Fanuc KAREL source: Client.kl

PROGRAM TCP_Client

------------------------------------ TCP_Client Plug-In ------------------------------------
-- Author: Niccolo' Quadrani
-- Date: 9/05/2025
-- Version: 1.0.0
------------------------------------ TCP_Client Plug-In ------------------------------------


------------------------------------ Import ------------------------------------

%RWACCESS
%STACKSIZE = 4096
%NOLOCKGROUP
%NOBUSYLAMP
%NOPAUSE = ERROR + COMMAND + TPENABLE
%ENVIRONMENT uif
%ENVIRONMENT sysdef
%ENVIRONMENT memo
%ENVIRONMENT kclop
%ENVIRONMENT bynam
%ENVIRONMENT fdev
%ENVIRONMENT flbt
%ENVIRONMENT regope
%ENVIRONMENT strng
%INCLUDE klevccdf
%INCLUDE klevkeys
%INCLUDE klevkmsk

------------------------------------ Variables Declaration ------------------------------------
VAR
    -- File variables (Used as a socket)
    f_socket:                        FILE

    -- Integers Variables
    i_debug:                        INTEGER
    i_command:                      INTEGER
    i_exe_flag:                     INTEGER
    i_object_number:                INTEGER
    i_status:                       INTEGER
    i_bytes_to_read:                INTEGER
    i_error:                        INTEGER

    -- Real Variables
    r_value:                        REAL

    -- Bolean Variables
    b_real_flag:                    BOOLEAN

    -- String variables
    s_send_command:                 STRING [64]
    s_custom_command:               STRING [64]
    s_received_string:              STRING [64]
    s_recipe:                       STRING [32]
    s_response:                     STRING [32]
    s_error:                        STRING [32]
    s_command:                      STRING [32]

    -- Integer Registers
    ir_i_debug_register:            INTEGER
    ir_i_command_register:          INTEGER
    ir_io_exe_register:             INTEGER
    ir_o_object_register:           INTEGER

    -- String Registers
    sr_i_custom_command:            INTEGER
    sr_io_recipe:                   INTEGER
    sr_o_response:                  INTEGER
    sr_o_error:                     INTEGER

    -- Position Registers
    pr_o_object_position:           INTEGER

------------------------------------ Debug Routine ------------------------------------
ROUTINE debug(s_msg:STRING)
VAR
    -- Used to format the debugs
    formatted_msg : STRING[64]

BEGIN
    -- Getting the register value
    GET_REG(ir_i_debug_register, b_real_flag, i_debug, r_value, i_status)

    IF i_status = 0 THEN -- Error check
        IF i_debug <> 0 THEN
            formatted_msg = 'DEBUG: ' + s_msg
            WRITE (formatted_msg, CR) -- Debugging on the CR
        ENDIF
    ELSE
        WRITE ('ERROR: Cannot execute GET_REG', CR) -- Printing the error in the CR
    ENDIF
END debug

------------------------------------ Registers Set-Up ------------------------------------
ROUTINE registers_setup(i_status:INTEGER)
BEGIN
    -- Setting-up the INTEGER registers
    ir_i_debug_register = 1
    ir_i_command_register = 2
    ir_io_exe_register = 3
    ir_o_object_register = 4

    -- Commenting the registers
    SET_REG_CMT (ir_i_debug_register,       'Activate debug', i_status)
    SET_REG_CMT (ir_i_command_register,     'Command', i_status)
    SET_REG_CMT (ir_io_exe_register,        'Execute', i_status)
    SET_REG_CMT (ir_o_object_register,      'Object number', i_status)

    -- Resetting the values of the registers
    SET_INT_REG (ir_i_debug_register,    0, i_status)
    SET_INT_REG (ir_i_command_register,  0, i_status)
    SET_INT_REG (ir_io_exe_register,    -1, i_status) -- Set to -1 to give a feedback on the connection, set to 0 after the connection
    SET_INT_REG (ir_o_object_register,   0, i_status)

    -- Setting-up the STRING registers
    sr_i_custom_command = 1
    sr_io_recipe = 2
    sr_o_response = 3
    sr_o_error = 4

    -- Commenting the registers
    SET_SREG_CMT (sr_i_custom_command,       'Custom command', i_status)
    SET_SREG_CMT (sr_io_recipe,              'Recipe name', i_status)
    SET_SREG_CMT (sr_o_response,             'Vision response', i_status)
    SET_SREG_CMT (sr_o_error,                'Vision error', i_status)

    -- Resetting the values of the registers
    SET_STR_REG (sr_i_custom_command,   '', i_status)
    SET_STR_REG (sr_io_recipe,          '', i_status)
    SET_STR_REG (sr_o_response,         '', i_status)
    SET_STR_REG (sr_o_error,            '', i_status)

    -- Setting-up the POSITION registers
    pr_o_object_position = 1

    -- Commenting the registers
    SET_PREG_CMT (pr_o_object_position, 'Vision coordinates', i_status)
END registers_setup

------------------------------------ Getting the command from the integer value  -----------------------------------
ROUTINE get_command(i_command:INTEGER)
BEGIN
    IF ((i_command > 0) AND (i_command < 8)) THEN

        IF  i_command = 1 THEN
                s_command = 'start_vision'
            ENDIF

            IF  i_command = 2 THEN
                s_command = 'stop_vision'
            ENDIF

            IF  i_command = 3 THEN
                s_command = 'locate'
            ENDIF

            IF  i_command = 4 THEN
                s_command = 'get_recipe'
            ENDIF

            IF  i_command = 5 THEN
                GET_STR_REG(sr_io_recipe, s_recipe, i_status) -- Getting the recipe name to load
                s_command = 'set_Recipe = ' + s_recipe -- String concatenation
            ENDIF

            IF  i_command = 6 THEN
                s_command = 'state'
            ENDIF

            IF  i_command = 7 THEN
                GET_STR_REG(sr_i_custom_command, s_custom_command, i_status) -- Getting the custom command to execute
                s_command = s_custom_command -- Formatting the command
            ENDIF

    ELSE
        i_command = -1 -- Command selected error
    ENDIF
END get_command

------------------------------------ Getting the command from the integer value  -----------------------------------
ROUTINE connection_init (client:STRING)
BEGIN
    -- Connecting to the client before doing any client related operation
    MSG_CONNECT(client,i_status)
    WHILE i_status <> 0 DO
        CLR_IO_STAT(f_socket) -- Clearing the IO status from older runs
        MSG_DISCO(client,i_status) -- Clearing the socket connection
        DELAY(100)
        MSG_CONNECT(client,i_status)
    ENDWHILE

    OPEN FILE f_socket ('rw',client) -- Opening the file using write mode on client 3
    i_status = IO_STATUS(f_socket) -- Checking the current IO i_status

    WHILE i_status <> 0 DO -- Looping until the socket file is open
        CLOSE FILE f_socket -- Closing the file to reset the connection
        DELAY(50) -- Waiting for the connection to be established
        OPEN FILE f_socket ('rw',client) -- Opening the file using write mode on client 3
        DELAY(25)
        i_status = IO_STATUS(f_socket) -- Checking the current IO i_status
    ENDWHILE

    -- Cleaning the file buffer
    BYTES_AHEAD(f_socket,i_bytes_to_read,i_status) -- Reading if there are any remained data
    IF i_bytes_to_read >= 1 THEN
        READ f_socket (s_received_string::i_bytes_to_read)
    ENDIF
    SET_INT_REG (ir_io_exe_register, 0, i_status) -- Connection ok feed back
END connection_init

------------------------------------ MAIN ------------------------------------
BEGIN
    registers_setup(i_status)
    debug('Registers setted-up')
    connection_init('C3:') -- Client used in the comunication

    -- Main cicle
     WHILE TRUE DO -- Looping until the socket file is open
        -- Waiting for the execute command
        REPEAT
            GET_REG(ir_io_exe_register, b_real_flag, i_exe_flag, r_value, i_status) -- Getting the execution register value
            DELAY(50)
        UNTIL ((i_exe_flag = 0) OR (i_exe_flag = -1)) -- Case "No exe" or "Error"

        GET_REG(ir_i_command_register, b_real_flag, i_command, r_value, i_status) -- Getting the command to send to the vision server

        get_command(i_command)

        IF i_command = -1 THEN
            debug('The selected command does not exist, please choose a command between 1 and 7')
            SET_STR_REG (sr_o_error, 'No valid command', i_status)
            SET_INT_REG (ir_io_exe_register, -1, i_status)
            GO TO skip_iteration -- Like a continue in the loop, jumping to the skip_iteration lable
        ENDIF

        WRITE f_socket(s_command) -- Sending the command to the vision server using the file socket
        SET_INT_REG (ir_i_command_register, 0, i_status) -- Setting the command register to 0 to reset it

        -- Reading the response from the vision server
        REPEAT
            BYTES_AHEAD(f_socket ,i_bytes_to_read,i_status)
            DELAY(50)
        UNTIL (i_bytes_to_read <= 0)

        READ f_socket (s_received_string::i_bytes_to_read) -- Reading the response

        IF i_command = 3 THEN
            -- Splitting the coordinates

        ELSE
            i_error = INDEX(s_received_string, '#') -- Checking if the char "#" is present in the string to launch an error

            IF i_error <> 0 THEN
                SET_STR_REG (sr_o_error, 'Error from the vision server', i_status) -- Writing the error in the error register
                SET_INT_REG (ir_io_execute_register, -1, i_status) -- Writing the error ack in the register
                debug(s_received_string) -- Printing the error string
                GO TO skip_iteration -- Skipping the iteration
            ELSE
                -- Setting string registers
                debug(s_received_string)
                SET_STR_REG (sr_o_response, s_received_string, i_status)
            ENDIF
        ENDIF

        SET_INT_REG (ir_io_exe_register, 0, i_status) -- Command ended
        SET_STR_REG (sr_o_error, '', i_status) -- Resetting the error
        i_bytes_to_read = 0
        s_received_string = ''

        skip_iteration:: -- Continue lable
    ENDWHILE
END TCP_Client
